// TIA Portal V18 export
FUNCTION "AHURegsCtrl_1" : Void   // FC60035, LAD
{ S7_Optimized_Access := 'TRUE' }
VERSION : 0.1
// Operation Modes                                                 Unit State
// 0=Protection                                                         0=Stopped
// 1=Economy                                                           1=Checking-up  
// 2=PreComfort                                                       2=Preheating
// 3=Comfor                                                              3=Starting 
// 4=Auto(Scheduler)                                              4=RecirculatingOperation (Protection)
//                                                                                 5=Sustained Mode (Economy setpoints)
//                                                                                 6=Sustained Mode (PreComfort setpoints) 
//                                                                                 7=Comfort  operation
//                                                                                 8=Stopping
//                                                                                 9=Blocking
// stored: AutoNumber false, IsIECCheckEnabled false, SetENOAutomatically false, UDAEnableTagReadback false
   VAR_INPUT
      iUnitID : Int;
      cActualOpMode : Byte;
      cHeatingRegCfg : Byte;
      cCoolingRegCfg : Byte;
      cIAQRegCfg : Byte;
      cBuildingdPRegCfg : Byte;
      xOtherBlockingAlarm : Bool;
      xFrostProtBlocking : Bool;
   END_VAR
   VAR_OUTPUT
      cTargetState : Byte;
      cHeatingRegState : Byte;
      cCoolingRegState : Byte;
      cIAQRegState : Byte;
      cBuildingdPRegState : Byte;
   END_VAR
   VAR_TEMP
      cActualOpModeSequence : Byte;   // Поточний цикл
   END_VAR
BEGIN

REGION Network 1 (SCL)
   IF #xFrostProtBlocking THEN
       // Frost protection
       #cTargetState := 11;
   ELSIF #xOtherBlockingAlarm THEN
       // Blocking Alarm
       #cTargetState := 10;
   ELSE
       CASE #cActualOpMode OF
           0:  // Protection 
               "AHURegsAndTargetStatesInProtectionOpMode"(iUnitID:=#iUnitID,
                                                          cActualOpMode:=#cActualOpMode,
                                                          cHeatingRegCfg:=#cHeatingRegCfg,
                                                          cCoolingRegCfg:=#cCoolingRegCfg,
                                                          cIAQRegCfg:=#cIAQRegCfg,
                                                          cBuildingdPRegCfg:=#cBuildingdPRegCfg,
                                                          cTargetState=>#cTargetState,
                                                          cHeatingRegState=>#cHeatingRegState,
                                                          cCoolingRegState=>#cCoolingRegState,
                                                          cIAQRegState=>#cIAQRegState,
                                                          cBuildingdPRegState=>#cBuildingdPRegState);

           1:  // Economy
               "AHURegsAndTargetStatesInEconomyOpMode"(iUnitID:=#iUnitID,
                                                       cActualOpMode:=#cActualOpMode,
                                                       cHeatingRegCfg:=#cHeatingRegCfg,
                                                       cCoolingRegCfg:=#cCoolingRegCfg,
                                                       cIAQRegCfg:=#cIAQRegCfg,
                                                       cBuildingdPRegCfg:=#cBuildingdPRegCfg,
                                                       cTargetState=>#cTargetState,
                                                       cHeatingRegState=>#cHeatingRegState,
                                                       cCoolingRegState=>#cCoolingRegState,
                                                       cIAQRegState=>#cIAQRegState,
                                                       cBuildingdPRegState=>#cBuildingdPRegState);
           2: // PreComfort
               "AHURegsAndTargetStatesInPreComfortOpMode"(iUnitID:=#iUnitID,
                                                          cActualOpMode:=#cActualOpMode,
                                                          cHeatingRegCfg:=#cHeatingRegCfg,
                                                          cCoolingRegCfg:=#cCoolingRegCfg,
                                                          cIAQRegCfg:=#cIAQRegCfg,
                                                          cBuildingdPRegCfg:=#cBuildingdPRegCfg,
                                                          cTargetState=>#cTargetState,
                                                          cHeatingRegState=>#cHeatingRegState,
                                                          cCoolingRegState=>#cCoolingRegState,
                                                          cIAQRegState=>#cIAQRegState,
                                                          cBuildingdPRegState=>#cBuildingdPRegState);
           ELSE  //Comfort
               "AHURegsAndTargetStatesInComfortOpMode"(iUnitID:=#iUnitID,
                                                       cActualOpMode:=#cActualOpMode,
                                                       cHeatingRegCfg:=#cHeatingRegCfg,
                                                       cCoolingRegCfg:=#cCoolingRegCfg,
                                                       cIAQRegCfg:=#cIAQRegCfg,
                                                       cBuildingdPRegCfg:=#cBuildingdPRegCfg,
                                                       cTargetState=>#cTargetState,
                                                       cHeatingRegState=>#cHeatingRegState,
                                                       cCoolingRegState=>#cCoolingRegState,
                                                       cIAQRegState=>#cIAQRegState,
                                                       cBuildingdPRegState=>#cBuildingdPRegState);
       END_CASE;
       ;
   END_IF;
END_REGION
END_FUNCTION
